{attribute 'no_explicit_call' := 'do not call this POU directly'}
FUNCTION_BLOCK INTERNAL FINAL FB_TestSuiteNameProvider IMPLEMENTS I_TestFrameWorkAdapter
VAR_INPUT
END_VAR
VAR_OUTPUT
END_VAR
VAR
	sTestSuiteNameField 	: T_MaxString;
	sTestNameField			: T_MaxString;
END_VAR

METHOD INTERNAL SetTestNames
VAR_INPUT CONSTANT
	sTestSuiteName 	: REFERENCE TO T_MaxString;
	sTestName		: REFERENCE TO T_MaxString;
END_VAR

sTestSuiteNameField := sTestSuiteName;
sTestNameField := sTestName;
END_METHOD

PROPERTY sTestName : REFERENCE TO Tc2_System.T_MaxString
GET
sTestName REF= sTestNameField;
END_GET
END_PROPERTY

PROPERTY sTestSuiteName : REFERENCE TO Tc2_System.T_MaxString
GET
sTestSuiteName REF= sTestSuiteNameField;
END_GET
END_PROPERTY

METHOD Verify : HRESULT
VAR_INPUT
	{attribute 'analysis' := '-33'}
	anyArg	: __SYSTEM.AnyType;
END_VAR
Verify := Tc2_System.E_HRESULTAdsErr.ACCESSDENIED;
END_METHOD

END_FUNCTION_BLOCK

(* stored: Version 1.1.0.1, ProductVersion 3.1.4026.18
   POU FB_TestSuiteNameProvider: Id {1618468c-8e9f-47a1-883e-b9b76a908690}, SpecialFunc None
   Method SetTestNames: Id {59071bf7-e632-4d90-9a60-a1aa486f91f4}
   Property sTestName: Id {f298cfe5-47f2-41ea-8807-db37151db457}
   Get Get: Id {aa8f7eee-3227-412c-a6da-09e65606d4d5}
   Property sTestSuiteName: Id {33a02c3b-8305-4a26-abb4-e397c7f1ca76}
   Get Get: Id {27aa5c98-63ed-4fa9-9d95-d2d0db9665c8}
   Method Verify: Id {38caa7fa-54bf-48d1-9737-a24c040eb1de} *)
